(* PLC project DCmotormechanic, Dassault Systèmes orchideo | easySSP (eXXcellent solutions GmbH) orchideo | easySSP (eXXcellent solutions GmbH) *)
(* stored: creationDateTime 2024-02-06T13:21:37Z, contentDescription DC-motor-mechanic.ssd *)

FUNCTION_BLOCK edrive_mass
  VAR_INPUT
    M_A : REAL := 0.0;
    M_B : REAL := 0.0;
  END_VAR
  VAR_OUTPUT
    wA : REAL := 0.0;
    wB : REAL := 0.0;
    phiB : REAL := 0.0;
    phiA : REAL := 0.0;
  END_VAR


ACTION C_source_code:

END_ACTION
END_FUNCTION_BLOCK

FUNCTION_BLOCK stimuli_model
  VAR_OUTPUT
    M_load : REAL := 0.0;
    U : REAL := 0.0;
  END_VAR


ACTION C_source_code:

END_ACTION
END_FUNCTION_BLOCK

PROGRAM DCmotormechanic.DCmotormechanic
  VAR_OUTPUT
    M : REAL := 0.0;
    wB : REAL := 0.0;
  END_VAR

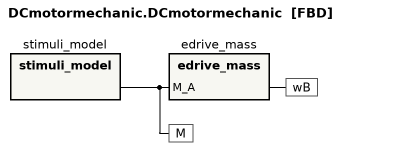
(* FBD diagram, written out as Structured Text *)
stimuli_model();
M := stimuli_model.M_load;
edrive_mass(M_A := stimuli_model.M_load);
wB := edrive_mass.wB;
END_PROGRAM
